FUNCTION_BLOCK FB_GCM
VAR_IN_OUT
	stVG	:	ST_VG;
END_VAR
VAR_OUTPUT
END_VAR
VAR
	rMinPressure: REAL;
	rV	:REAL;
END_VAR

(* Baratron Pressure Calc 
A. Wallace
2016-6-16
The full-scale pressure times the ratio of the meas.
voltage to full-scale voltage (10V).
The minimum pressure is always going to be 5e-4 * F.S.V.*)

rMinPressure := stVG.rFULL_SCALE * 5E-4;


rV :=MAX((10*INT_TO_REAL(stVG.iPRESS_R)/32767),0);
stVG.rPRESS := (stVG.rFULL_SCALE/10)*rV;
IF stVG.rPRESS > rMinPressure THEN
	stVG.xPRESS_OK := TRUE;
ELSE
	stVG.xPRESS_OK := FALSE;
END_IF

END_FUNCTION_BLOCK

(* stored: Version 1.1.0.1, ProductVersion 3.1.4018.5
   POU FB_GCM: Id {d03d0435-a8a4-4ab2-9d39-a304a183952d}, SpecialFunc None *)
